(* IEC 61131-3 sources: Hal/Libraries/CAN_Lib, 3 files *)

(* ---- CAN_Lib.typ ---- *)
(********************************************************************
 * COPYRIGHT -- Bernecker + Rainer
 ********************************************************************
 * Library: CAN_Lib
 * File: CAN_Lib.typ
 * Author: B+R
 ********************************************************************
 * Data types of library CAN_Lib
 ********************************************************************)

TYPE
	INFO_typ : STRUCT				(*CAN statistic data*)
		received	: UDINT ;		(*the sum of all received CAN frames*)
		transmit	: UDINT ;		(*the sum of all sent CAN frames*)
		error	: UDINT ;			(*the sum of all error messages from the CAN device*)
		busoff	: UDINT ;			(*the sum of all CAN BusOff errors*)
		warning	: UDINT ;			(*the sum of all CAN warning errors*)
		other	: UDINT ;			(*the sum of other errors*)
		lost	: UDINT ;			(*the sum of all overwritten CAN frames*)
		stufferror	: UDINT ;		(*the sum of stuff errors*)
		formerror	: UDINT ;		(*the sum of form errors*)
		ackerror	: UDINT ;		(*the sum of ack errors*)
		bit1error	: UDINT ;		(*the sum of bit1 errors*)
		bit0error	: UDINT ;		(*the sum of bit0 errors*)
		crcerror	: UDINT ;		(*the sum of crc errors*)
		lec0	: UDINT ;			(*the sum of all errors with Last Error Code=0*)
		rxirq	: UDINT ;			(*the sum of all received interrupts*)
		txirq	: UDINT ;			(*the sum of all sent interrupts*)
	END_STRUCT;
	DevParam : STRUCT				(*points to the DeviceParameter structure*)
		baudrate	: USINT ;		(*baud rate for the CAN controller to be opened*)
		cob_nr	: UINT ;			(*number of communication objects*)
		pError	: UDINT ;			(*address of / pointer to the error variable*)
		pDevice	: UDINT ;			(*address of / pointer to the DeviceString*)
		info	: UINT ;			(*bit 7 = 1 enables extended mode for the controller*)
	END_STRUCT;
END_TYPE

(* ---- CAN_Lib.fun ---- *)
(********************************************************************
 * COPYRIGHT -- Bernecker + Rainer
 ********************************************************************
 * Library: CAN_Lib
 * File: CAN_Lib.fun
 * Author: B+R
 ********************************************************************
 * Functions and function blocks of library CAN_Lib
 ********************************************************************)

FUNCTION_BLOCK CANinfo			(*reads the statistical data from a CAN device*)
	VAR_INPUT
		enable	:BOOL;			(*enables execution*)
		us_ident	:UDINT;		(*us_ident identifier from CANopen*)
		info_adr	:UDINT;		(*pointer to the CANinfo structure INFO_typ*)
	END_VAR
	VAR_OUTPUT
		status	:UINT;			(*execution status: ERR_OK, ERR_FUB_ENABLE_FALSE, 0xXXXX = see help*)
	END_VAR
END_FUNCTION_BLOCK

FUNCTION_BLOCK CANMulQueue		(*installs a queue for multiple CAN identifiers in the read direction*)
	VAR_INPUT
		enable	:BOOL;			(*enables execution*)
		us_ident	:UDINT;		(*us_ident from CANopen / CANMulOpen*)
		pCAN_id	:UDINT;			(*pointer to an array of CAN identifiers*)
		ID_nr	:USINT;			(*number of CAN identifiers*)
		size	:UINT;			(*number of telegrams in the queue*)
	END_VAR
	VAR_OUTPUT
		q_ident	:UDINT;			(*identifier for CANmulrd*)
		status	:UINT;			(*execution status: ERR_OK, ERR_FUB_ENABLE_FALSE, 0xXXXX = see help*)
	END_VAR
	VAR
		old_enable	:BOOL;		(*internal variable*)
		cob_handle	:UDINT;		(*internal variable*)
		init_cnt	:UDINT;		(*internal variable*)
	END_VAR
END_FUNCTION_BLOCK

FUNCTION_BLOCK CANxMulQueue		(*installs a queue for multiple CAN identifiers in the read direction*)
	VAR_INPUT
		enable	:BOOL;			(*enables execution*)
		us_ident	:UDINT;		(*us_ident from CANopen / CANMulOpen*)
		pCAN_id	:UDINT;			(*pointer to an array of CAN identifiers*)
		ID_nr	:UDINT;			(*number of CAN identifiers*)
		size	:UINT;			(*number of telegrams in the queue*)
	END_VAR
	VAR_OUTPUT
		q_ident	:UDINT;			(*identifier for CANmulrd*)
		status	:UINT;			(*execution status: ERR_OK, ERR_FUB_ENABLE_FALSE, 0xXXXX = see help*)
	END_VAR
	VAR
		old_enable	:BOOL;		(*internal variable*)
		cob_handle	:UDINT;		(*internal variable*)
		init_cnt	:UDINT;		(*internal variable*)
	END_VAR
END_FUNCTION_BLOCK

FUNCTION_BLOCK CANMulOpen		(*initializes numerous CAN controllers and allocates the appropriate resources*)
	VAR_INPUT
		enable	:BOOL;			(*enables execution*)
		pDevParam	:UDINT;		(*pointer to the DeviceParameter structure*)
		dev_nr	:USINT;			(*number of CAN controllers to be opened*)
	END_VAR
	VAR_OUTPUT
		us_ident	:UDINT;		(*identifier for all additional CAN function blocks*)
		status	:UINT;			(*execution status: ERR_OK, ERR_FUB_ENABLE_FALSE, 0xXXXX = see help*)
	END_VAR
	VAR
		old_enable	:BOOL;		(*internal variable*)
		init_cnt	:UDINT;		(*internal variable*)
	END_VAR
END_FUNCTION_BLOCK

FUNCTION_BLOCK CANMulrd			(*copies data from the queue to the buffer or sends an error in the status*)
	VAR_INPUT
		enable	:BOOL;			(*enables execution*)
		q_ident	:UDINT;			(*identifier q_ident from CANMulQueue*)
		data_adr	:UDINT;		(*CAN data*)
	END_VAR
	VAR_OUTPUT
		size	:UINT;			(*length of the data*)
		ID	:UDINT;				(*CAN identifier which received the data*)
		status	:UINT;			(*execution status: ERR_OK, ERR_FUB_ENABLE_FALSE, 0xXXXX = see help*)
	END_VAR
END_FUNCTION_BLOCK

FUNCTION_BLOCK CANTime			(*reads the time stamp for a CAN object*)
	VAR_INPUT
		enable		:BOOL;		(*enables execution*)
		us_ident	:UDINT;		(*user ident from CANopen() / CANMulOpen()*)
		can_id	:UDINT;			(*CAN identifier*)
		pSystemTick	:UDINT;		(*pointer to the SystemTick counter*)
		pSystemStamp	:UDINT;	(*pointer to the SystemStamp*)
	END_VAR
	VAR_OUTPUT
		status	:UINT;			(*execution status: ERR_OK, ERR_FUB_ENABLE_FALSE, 0xXXXX = see help*)
	END_VAR
	VAR
		old_enable	:BOOL;		(*internal variable*)
		old_id	:UDINT;			(*internal variable*)
		cob_handle	:UDINT;		(*internal variable*)
	END_VAR
END_FUNCTION_BLOCK

FUNCTION_BLOCK CANquwr			(*sends a CAN message with the given CAN identifier to the CAN controller for transmission*)
	VAR_INPUT
		enable	:BOOL;			(*enables execution*)
		us_ident	:UDINT;		(*user ident number from the CANopen() function*)
		can_id	:UDINT;			(*CAN identifier*)
		data_adr	:UDINT;		(*address of the CAN data (max. 8 bytes)*)
		data_lng	:USINT;		(*length of the data (max. 8 bytes)*)
	END_VAR
	VAR_OUTPUT
		status	:UINT;			(*execution status: ERR_OK, ERR_FUB_ENABLE_FALSE, 0xXXXX = see help*)
	END_VAR
	VAR
		old_enable	:BOOL;		(*internal variable*)
		cob_handle	:UDINT;		(*internal variable*)
		init_cnt	:UDINT;		(*internal variable*)
	END_VAR
END_FUNCTION_BLOCK

FUNCTION_BLOCK SetNdNr			(*saves the transferred node number and device description in the CRM*)
	VAR_INPUT
		enable	:BOOL;			(*enables execution*)
		device	:UDINT;			(*pointer to a string containing the device description, e.g. "SLx.SSx.IFx"*)
		nodenr	:USINT;			(*new node number*)
	END_VAR
	VAR_OUTPUT
		status	:UINT;			(*execution status: ERR_OK, ERR_FUB_ENABLE_FALSE, 0xXXXX = see help*)
	END_VAR
END_FUNCTION_BLOCK

FUNCTION_BLOCK GetNdNr			(*reads the stored node number and device description from the CRM*)
	VAR_INPUT
		enable	:BOOL;			(*enables execution*)
		dev_adr	:UDINT;			(*pointer to a string containing the device description, e.g. "SLx.SSx.IFx"*)
	END_VAR
	VAR_OUTPUT
		nodenr	:USINT;			(*the node number read from the CRM*)
		status	:UINT;			(*execution status: ERR_OK, ERR_FUB_ENABLE_FALSE, 0xXXXX = see help*)
	END_VAR
END_FUNCTION_BLOCK

FUNCTION_BLOCK CMSexit			(*free the ressources of the list of CMS objects defined with the CMSinit() function*)
	VAR_INPUT
		enable	:BOOL;			(*enables execution*)
		cms_ident	:UDINT;		(*CMS identifier from CMSinit()*)
	END_VAR
	VAR_OUTPUT
		status	:UINT;			(*execution status: ERR_OK, ERR_FUB_ENABLE_FALSE, 0xXXXX = see help*)
	END_VAR
END_FUNCTION_BLOCK

FUNCTION_BLOCK CMSmain			(*edits the list of CMS objects defined with the CMSinit() function*)
	VAR_INPUT
		enable	:BOOL;			(*enables execution*)
		cms_ident	:UDINT;		(*CMS identifier from CMSinit()*)
		cms_mode	:UDINT;		(*2 ... WRITE, send/update data*)
	END_VAR
	VAR_OUTPUT
		status	:UINT;			(*execution status: ERR_OK, ERR_FUB_ENABLE_FALSE, 0xXXXX = see help*)
	END_VAR
	VAR
		init_cnt	:UDINT;		(*internal variable*)
	END_VAR
END_FUNCTION_BLOCK

FUNCTION_BLOCK CMSinit			(*sends and receives CMS objects*)
	VAR_INPUT
		enable	:BOOL;			(*enables execution*)
		us_ident	:UDINT;		(*user ident from CANopen()*)
		user_type	:USINT;		(*0 CLIENT node type, 1 SERVER node type*)
		queue_cnt	:UINT;		(*reserved*)
		modul_name	:UDINT;		(*pointer to the string containing the name of the data object*)
	END_VAR
	VAR_OUTPUT
		cms_entry	:UINT;		(*error entry number or number of CMS objects in the CMS data object*)
		cms_ident	:UDINT;		(*CMS identifier is needed for CMSmain()*)
		status	:UINT;			(*execution status: ERR_OK, ERR_FUB_ENABLE_FALSE, 0xXXXX = see help*)
	END_VAR
	VAR
		old_enable	:BOOL;		(*internal variable*)
		init_cnt	:UDINT;		(*internal variable*)
	END_VAR
END_FUNCTION_BLOCK

FUNCTION_BLOCK CMSdlreq			(*transfers a "multiplexed domain" object of any data size from the client to the server*)
	VAR_INPUT
		enable	:BOOL;			(*enables execution*)
		initiate	:BOOL;		(*pos. edge (0->1) ... Initiate new domain*)
		us_ident	:UDINT;		(*user ID from CANopen()*)
		client_id	:UDINT;		(*CAN identifier for the send COB from client to server*)
		server_id	:UDINT;		(*CAN identifier for the send COB from server to client*)
		mult	:UDINT;			(*multiplexer for multiplexed domain*)
		data_adr	:UDINT;		(*address of the download data*)
		data_len	:UDINT;		(*length of the download data*)
	END_VAR
	VAR_OUTPUT
		add_code	:UINT;		(*additional error information in the event of abnormal termination*)
		err_class	:USINT;		(*error class according to CANopen()*)
		err_code	:USINT;		(*error according to CANopen()*)
		dl_len	:UDINT;			(*size of the download data sent*)
		status	:UINT;			(*execution status: ERR_OK, ERR_FUB_ENABLE_FALSE, 0xXXXX = see help*)
	END_VAR
	VAR
		cob_handle	:UDINT;		(*internal variable*)
		init_cnt	:UDINT;		(*internal variable*)
		old_enable	:BOOL;		(*internal variable*)
	END_VAR
END_FUNCTION_BLOCK

FUNCTION_BLOCK CMSdlcon			(*enables a "multiplexed domain" object of any data length to be received by the server*)
	VAR_INPUT
		enable	:BOOL;			(*enables execution*)
		initiate	:BOOL;		(*1 ... startpulse, activation receiving the domain*)
		us_ident	:UDINT;		(*user ID from CANopen()*)
		client_id	:UDINT;		(*CAN identifier for the send COB from client to server*)
		server_id	:UDINT;		(*CAN identifier for the send COB from server to client*)
		data_adr	:UDINT;		(*address of the download data*)
		data_len	:UDINT;		(*length of the download data in bytes*)
	END_VAR
	VAR_OUTPUT
		add_code	:UINT;		(*additional error information in the event of abnormal termination*)
		err_class	:USINT;		(*error class according to CANopen()*)
		err_code	:USINT;		(*error according to CANopen()*)
		mult	:UDINT;			(*multiplexer for multiplexed domain*)
		dl_len	:UDINT;			(*size of the data already downloaded*)
		status	:UINT;			(*execution status: ERR_OK, ERR_FUB_ENABLE_FALSE, 0xXXXX = see help*)
	END_VAR
	VAR
		old_enable	:BOOL;		(*internal variable*)
		cob_handle	:UDINT;		(*internal variable*)
		init_cnt	:UDINT;		(*internal variable*)
	END_VAR
END_FUNCTION_BLOCK

FUNCTION_BLOCK CANxnode			(*determines the node number set with the x-th CAN node switch*)
	VAR_INPUT
		enable	:BOOL;			(*enables execution*)
		us_ident	:UDINT;		(*user Ident from CANopen()*)
	END_VAR
	VAR_OUTPUT
		node_nr	:USINT;			(*node number of the CAN station (0x00 through 0xFF)*)
		status	:UINT;			(*execution status: ERR_OK, ERR_FUB_ENABLE_FALSE, 0xXXXX = see help*)
	END_VAR
END_FUNCTION_BLOCK

FUNCTION_BLOCK CANwrite			(*sends a CAN message with the given CAN identifier to the CAN controller for transmission*)
	VAR_INPUT
		enable	:BOOL;			(*enables execution*)
		us_ident	:UDINT;		(*user ident number from the CANopen() function*)
		can_id	:UDINT;			(*CAN identifier*)
		data_adr	:UDINT;		(*address of the CAN data (max. 8 bytes)*)
		data_lng	:USINT;		(*length of the data (max. 8 bytes)*)
	END_VAR
	VAR_OUTPUT
		status	:UINT;			(*execution status: ERR_OK, ERR_FUB_ENABLE_FALSE, 0xXXXX = see help*)
	END_VAR
	VAR
		old_enable	:BOOL;		(*internal variable*)
		old_id	:UDINT;			(*internal variable*)
		cob_handle	:UDINT;		(*internal variable*)
		init_cnt	:UDINT;		(*internal variable*)
		wr_order	:USINT;		(*internal variable*)
		align_byte	:USINT;		(*internal variable*)
	END_VAR
END_FUNCTION_BLOCK

FUNCTION_BLOCK CANupd			(*gives the response to an RTR request telegram to the send node*)
	VAR_INPUT
		enable	:BOOL;			(*enables execution*)
		us_ident	:UDINT;		(*user ident from CANopen()*)
		can_id	:UDINT;			(*CAN identifier*)
		data_adr	:UDINT;		(*address of the data area in which the update data is stored*)
		data_lng	:USINT;		(*length of the update data in bytes*)
	END_VAR
	VAR_OUTPUT
		status	:UINT;			(*execution status: ERR_OK, ERR_FUB_ENABLE_FALSE, 0xXXXX = see help*)
	END_VAR
	VAR
		old_enable	:BOOL;		(*internal variable*)
		old_id	:UDINT;			(*internal variable*)
		cob_handle	:UDINT;		(*internal variable*)
		init_cnt	:UDINT;		(*internal variable*)
	END_VAR
END_FUNCTION_BLOCK

FUNCTION_BLOCK CANngp			(*handles the Node Guarding Protocol according to CAL on the NMT slave*)
	VAR_INPUT
		enable	:BOOL;			(*enables execution*)
		us_ident	:UDINT;		(*user ident from CANopen()*)
		can_id	:UDINT;			(*CAN identifier*)
		nd_state	:USINT;		(*node status*)
	END_VAR
	VAR_OUTPUT
		status	:UINT;			(*execution status: ERR_OK, ERR_FUB_ENABLE_FALSE, 0xXXXX = see help*)
	END_VAR
	VAR
		old_enable	:BOOL;		(*internal variable*)
		old_id	:UDINT;			(*internal variable*)
		cob_handle	:UDINT;		(*internal variable*)
		init_cnt	:UDINT;		(*internal variable*)
	END_VAR
END_FUNCTION_BLOCK

FUNCTION_BLOCK CANrwtab			(*edits the list of variables (variables table) defined with the CANdftab()*)
	VAR_INPUT
		enable	:BOOL;			(*enables execution*)
		tab_ident	:UDINT;		(*table identifier from CANdftab()*)
	END_VAR
	VAR_OUTPUT
		status	:UINT;			(*execution status: ERR_OK, ERR_FUB_ENABLE_FALSE, 0xXXXX = see help*)
	END_VAR
END_FUNCTION_BLOCK

FUNCTION_BLOCK CANrtr			(*sends an RTR request frame on the CAN bus*)
	VAR_INPUT
		enable	:BOOL;			(*enables execution*)
		request	:BOOL;			(*0 poll data buffer, 1 send RTR request*)
		us_ident	:UDINT;		(*user ident from CANopen()*)
		can_id	:UDINT;			(*CAN identifier*)
		data_adr	:UDINT;		(*address of the data area in which the data received is stored*)
	END_VAR
	VAR_OUTPUT
		data_lng	:USINT;		(*length of the received data in bytes*)
		status	:UINT;			(*execution status: ERR_OK, ERR_FUB_ENABLE_FALSE, 0xXXXX = see help*)
	END_VAR
	VAR
		old_enable	:BOOL;		(*internal variable*)
		cob_handle	:UDINT;		(*internal variable*)
		init_cnt	:UDINT;		(*internal variable*)
	END_VAR
END_FUNCTION_BLOCK

FUNCTION_BLOCK CANread			(*reads CAN messages from the CAN controller*)
	VAR_INPUT
		enable	:BOOL;			(*enables execution*)
		us_ident	:UDINT;		(*user ident number from the CANopen() function*)
		can_id	:UDINT;			(*CAN identifier*)
		data_adr	:UDINT;		(*address where the read data is stored (max. 8 bytes)*)
	END_VAR
	VAR_OUTPUT
		data_lng	:USINT;		(*length of the data*)
		status	:UINT;			(*execution status: ERR_OK, ERR_FUB_ENABLE_FALSE, 0xXXXX = see help*)
	END_VAR
	VAR
		old_enable	:BOOL;		(*internal variable*)
		cob_handle	:UDINT;		(*internal variable*)
		init_cnt	:UDINT;		(*internal variable*)
	END_VAR
END_FUNCTION_BLOCK

FUNCTION_BLOCK CANrd			(*copies data from the queue to the buffer or sends an error in the status*)
	VAR_INPUT
		enable	:BOOL;			(*enables execution*)
		q_ident	:UDINT;			(*queue identifier from CANqueue()*)
		data_adr	:UDINT;		(*address of the data area where CAN data from the receive queue is stored*)
	END_VAR
	VAR_OUTPUT
		size	:UINT;			(*length of the CAN data in bytes*)
		status	:UINT;			(*execution status: ERR_OK, ERR_FUB_ENABLE_FALSE, 0xXXXX = see help*)
	END_VAR
END_FUNCTION_BLOCK

FUNCTION_BLOCK CANxrd			(*copies data from the queue to the buffer or sends an error in the status*)
	VAR_INPUT
		enable	:BOOL;			(*enables execution*)
		q_ident	:UDINT;			(*queue identifier from CANqueue()*)
		data_adr	:UDINT;		(*address of the data area where CAN data from the receive queue is stored*)
	END_VAR
	VAR_OUTPUT
		can_id	:UDINT;			(*CAN identifier*)
		size	:UINT;			(*length of the CAN data in bytes*)
		status	:UINT;			(*execution status: ERR_OK, ERR_FUB_ENABLE_FALSE, 0xXXXX = see help*)
	END_VAR
END_FUNCTION_BLOCK

FUNCTION_BLOCK CANqueue			(*installs a queue for a CAN identifier in the read direction*)
	VAR_INPUT
		enable	:BOOL;			(*enables execution*)
		us_ident	:UDINT;		(*user Ident from CANopen()*)
		can_id	:UDINT;			(*CAN identifier for the queue*)
		size	:UINT;			(*number of telegrams in the queue*)
	END_VAR
	VAR_OUTPUT
		q_ident	:UDINT;			(*queue identifier for the CANrd()*)
		status	:UINT;			(*execution status: ERR_OK, ERR_FUB_ENABLE_FALSE, 0xXXXX = see help*)
	END_VAR
	VAR
		old_enable	:BOOL;		(*internal variable*)
		cob_handle	:UDINT;		(*internal variable*)
		init_cnt	:UDINT;		(*internal variable*)
	END_VAR
END_FUNCTION_BLOCK

FUNCTION_BLOCK CANopen			(*initializes the CAN controller and requests the necessary resources (e.g. memory)*)
	VAR_INPUT
		enable	:BOOL;			(*enables execution*)
		baud_rate	:USINT;		(*baud rate at which the CAN interface should be operated*)
		cob_anz	:UINT;			(*max. permissible number of COBs (communication objects)*)
		error_adr	:UDINT;		(*pointer to an error variable, e.g. Bit 15 = 1 the CAN bus is in the BusOff state*)
		device	:UDINT;			(*address of a string which clearly describes the CAN interface*)
		info	:UINT;			(*enables/disables extended mode for the CAN controller*)
	END_VAR
	VAR_OUTPUT
		us_ident	:UDINT;		(*is required for the other functions of the CAN_Lib library in order to identify a CAN interface clearly*)
		status	:UINT;			(*execution status: ERR_OK, ERR_FUB_ENABLE_FALSE, 0xXXXX = see help*)
	END_VAR
	VAR
		old_enable	:BOOL;		(*internal variable*)
		init_cnt	:UDINT;		(*internal variable*)
	END_VAR
END_FUNCTION_BLOCK

FUNCTION_BLOCK CANnode			(*determines the CAN node number*)
	VAR_INPUT
		enable	:BOOL;			(*enables execution*)
	END_VAR
	VAR_OUTPUT
		node_nr	:USINT;			(*node number of the CAN station (0x00 through 0xFF)*)
		status	:UINT;			(*execution status: ERR_OK, ERR_FUB_ENABLE_FALSE, 0xXXXX = see help*)
	END_VAR
END_FUNCTION_BLOCK

FUNCTION_BLOCK CANgetid			(*confirms the CAN identifier which the exception trigged in the context of an exception object*)
	VAR_INPUT
		enable	:BOOL;			(*enables execution*)
		data_adr	:UDINT;		(*address of the data area in which the data received is stored*)
	END_VAR
	VAR_OUTPUT
		data_lng	:USINT;		(*length of the received data in bytes*)
		can_id	:UDINT;			(*CAN identifier for the exception*)
		status	:UINT;			(*execution status: ERR_OK, ERR_FUB_ENABLE_FALSE, 0xXXXX = see help*)
	END_VAR
	VAR
		init_cnt	:UDINT;		(*internal variable*)
	END_VAR
END_FUNCTION_BLOCK

FUNCTION_BLOCK CANexcep			(*activates a pre-installed exception object with the exception number exc_no*)
	VAR_INPUT
		enable	:BOOL;			(*enables execution*)
		us_ident	:UDINT;		(*user Ident from CANopen()*)
		can_id	:UDINT;			(*CAN identifier*)
		exc_nr	:USINT;			(*number of the exception (exception numbers 208 to 223 are reserved for CAN)*)
	END_VAR
	VAR_OUTPUT
		status	:UINT;			(*execution status: ERR_OK, ERR_FUB_ENABLE_FALSE, 0xXXXX = see help*)
	END_VAR
	VAR
		old_enable	:BOOL;		(*internal variable*)
		init_cnt	:UDINT;		(*internal variable*)
		cob_handle	:UDINT;		(*internal variable*)
		ex_p	:UDINT;			(*internal variable*)
		ex_maxtask	:UDINT;		(*internal variable*)
		ss_irqvw_p	:UDINT;		(*internal variable*)
	END_VAR
END_FUNCTION_BLOCK

FUNCTION_BLOCK CANdftab			(*supplies a variables list (variables table) defined by the user with data about the CAN bus*)
	VAR_INPUT
		enable	:BOOL;			(*enables execution*)
		us_ident	:UDINT;		(*user ident number from the CANopen() function*)
		table_adr	:UDINT;		(*address of the variables table*)
		tab_num	:UINT;			(*number of entries in the variables table*)
	END_VAR
	VAR_OUTPUT
		tab_ident	:UDINT;		(*table identifier for CANrwtab()*)
		status	:UINT;			(*execution status: ERR_OK, ERR_FUB_ENABLE_FALSE, 0xXXXX = see help*)
	END_VAR
	VAR
		old_enable	:BOOL;		(*internal variable*)
		init_cnt	:UDINT;		(*internal variable*)
	END_VAR
END_FUNCTION_BLOCK

FUNCTION_BLOCK CANbtreg			(*configures a special bit timing register values for the CAN controller (Intel 82527)*)
	VAR_INPUT
		enable	:BOOL;			(*enables execution*)
		us_ident	:UDINT;		(*user Ident from CANopen()*)
		treg0	:UDINT;			(*bit timing register 0*)
		treg1	:UDINT;			(*bit timing Register 1*)
	END_VAR
	VAR_OUTPUT
		status	:UINT;			(*execution status: ERR_OK, ERR_FUB_ENABLE_FALSE, 0xXXXX = see help*)
	END_VAR
END_FUNCTION_BLOCK

(* ---- CAN_Lib.var ---- *)
(********************************************************************
 * COPYRIGHT (C) BERNECKER + RAINER, AUSTRIA, A-5142 EGGELSBERG
 ********************************************************************
 * Library: CAN_Lib
 * File: CAN_Lib.var
 * Created: 22.02.2010
 ********************************************************************
 * Constants of library CAN_Lib
 ********************************************************************)
VAR CONSTANT
	canERR_CAN_NOENTRY		: UINT	:= 8800;		(*not enough communication objects (COBs) available as specified in CANopen*)
	canERR_CAN_NOMEM		: UINT	:= 8801;		(*not enough memory available for resources*)
	canERR_CAN_WRIDENT		: UINT	:= 8802;		(*wrong identifier*)
	canERR_CAN_COBUSED		: UINT	:= 8803;		(*communication objects (COBs) identifier is already being used in the system*)
	canERR_CAN_WRCANID		: UINT	:= 8804;		(*wrong CAN identifier: Only standard CAN identifiers (11 bits) up to 2047 are permitted*)
	canERR_CAN_WRUSERID		: UINT	:= 8805;		(*incorrect user ID us_ident transferred, or the FBK cannot be used after a CANMulOpen*)
	canERR_CAN_COBDEF		: UINT	:= 8806;		(*a COB with the specified CAN identifier has already been defined in the system*)
	canERR_CAN_WRDEF		: UINT	:= 8807;		(*false CAN identifier definition*)
	canERR_CAN_WRHDLE		: UINT	:= 8808;		(*COB management (FBK memory) destroyed*)
	canERR_CAN_BUSY			: UINT	:= 8809;		(*CAN operation with the same CAN identifier is busy*)
	canERR_CAN_QFULL		: UINT	:= 8810;		(*transmit queue full*)
	canERR_CAN_BUSOFF		: UINT	:= 8811;		(*CAN bus is BusOff. Different baud rate on different nodes?*)
	canERR_CAN_NOHIGH		: UINT	:= 8812;		(*no more buffers available: All buffers (max. 13) in the can controller have already been defined and assigned*)
	canERR_CAN_NOTINST		: UINT	:= 8813;		(*CAN driver not installed: CAN2000.BR not loaded (needs to be transferred to target system)*)
	canERR_CAN_WRLNG		: UINT	:= 8814;		(*data type of event PV is not BYTES or the length of a write PV is greater than 8 bytes: CAN FBKs can only send data of length 8 bytes to the CAN bus*)
	canERR_CAN_BDRATE		: UINT	:= 8815;		(*illegal baud rate *)
	canERR_CAN_COBANZ		: UINT	:= 8816;		(*cob_anz in CANopen/CANMulOpen incorrect: cob_no must be less than 2048 and greater than 0*)
	canERR_CAN_NOCONTR		: UINT	:= 8817;		(*no CAN controller found: Error in the device string of the FBK CANopen / CANMulOpen or the CAN controller is not ready - hardware may not be present*)
	canERR_CAN_HTLXINF		: UINT	:= 8818;		(*error analyzing hardware*)
	canERR_CAN_HTLQUIT		: UINT	:= 8819;		(*error in interrupt handling*)
	canERR_CAN_NOFUNC		: UINT	:= 8820;		(*error in interrupt handling*)
	canERR_CAN_WRUSRTYP		: UINT	:= 8821;		(*user_typ in CMSinit is incorrect: user_typ must be 0 for client or 1 for server*)
	canERR_WRCMSOBJ			: UINT	:= 8822;		(*CMS object incorrectly defined: Syntax error in the CMS data object for CMSinit() (see cms_entry)*)
	canERR_CAN_WRSTRUCT		: UINT	:= 8823;		(*invalid CMS structure: The structure is too complex (only simple structures are permitted)*)
	canERR_CAN_WRMODE		: UINT	:= 8824;		(*incorrect value for cms_mode transferred to the CMSmain() function (valid value: 2)*)
	canERR_CAN_NO_NODE		: UINT	:= 8825;		(*node number cannot be read*)
	canERR_CAN_NILPTR		: UINT	:= 8826;		(*an invalid parameter has been transferred (NULL)*)
	canERR_CAN_IRQHANDLE	: UINT	:= 8827;		(*internal management is destroyed in the interrupt handler*)
	canERR_CAN_ABORTED		: UINT	:= 8828;		(*abort protocol has been sent to the client (>add_code)*)
	canERR_CAN_ABORTRECEIV	: UINT	:= 8829;		(*abort protocol has been received from the client*)
	canERR_CAN_FBHANDLE		: UINT	:= 8830;		(*incorrect FBCAN handle*)
	canERR_CAN_EXTENDED		: UINT	:= 8831;		(*conflict with standard/extended mode (11 or 29-bit CAN identifier): FBK configuration and system configuration (Automation Studio) of CAN interface do not match*)
	canERR_CMS_MULTIPLEX	: UINT	:= 8832;		(*CMS multiplexer definition error: Different object_typ, access_typ or ID or a multiplexer has been used more than once for an ID*)
	canERR_CAN_WROBJ		: UINT	:= 8833;		(*CAN object error: Tried to use a dynamic PV. Use a normal PV*)
	canERR_CAN_BITMODE		: UINT	:= 8834;		(*CAN identifier mode configured differently (11-bit / 29-bit, see the Automation Studio CAN device configuration)*)
	canERR_FBCAN_COB		: UINT	:= 8837;		(*INA2000 CAN: COB not defined*)
	canERR_FBCAN_NODENR		: UINT	:= 8838;		(*INA2000 CAN: Node number too large*)
	canERR_FBCAN_HANDLE		: UINT	:= 8839;		(*INA2000 CAN: Incorrect handle*)
	canERR_FBCAN_RXBUF		: UINT	:= 8840;		(*INA2000 CAN: No Rx buffer free*)
	canERR_CAN_STUFF		: UINT	:= 8841;		(*Warning: CAN: Stuff error -> CAN ID collision / baud rate*)
	canERR_CAN_FORM			: UINT	:= 8842;		(*Warning: CAN: Format error -> Baud rate*)
	canERR_CAN_ACK			: UINT	:= 8843;		(*Warning: CAN: ACK error - No acknowledge from other nodes*)
	canERR_CAN_BIT1			: UINT	:= 8844;		(*Warning: CAN: Bit1 send error (recessive bit)*)
	canERR_CAN_BIT0			: UINT	:= 8845;		(*Warning: CAN: Bit0 send error (dominant bit)*)
	canERR_CAN_CRC			: UINT	:= 8846;		(*Warning: CAN: CRC checksum error*)
	canERR_WRONG_OBJNR		: UINT	:= 8850;		(*CAN CCI: Object number not within value range*)
	canERR_NO_INIT_STATE	: UINT	:= 8851;		(*CAN CCI: Error during initialization*)
	canERR_NO_BUSOFF_STATE	: UINT	:= 8852;		(*CAN CCI: BUS_OFF problem*)
	canERR_NO_BUFFER_CFG	: UINT	:= 8853;		(*CAN CCI: Buffer not configured*)
	canERR_HW_RESET_ACTIVE	: UINT	:= 8854;		(*CAN CCI: Hardware in reset state*)
	canERR_CPU_UPDATE		: UINT	:= 8855;		(*CAN CCI: Error updating data*)
	canERR_OBJ_ACTIVE		: UINT	:= 8856;		(*CAN CCI: Buffer being processed*)
	canERR_READ_ONLY_OBJ	: UINT	:= 8857;		(*CAN CCI: Read-only object*)
	canERR_WRONG_CAN_MODE	: UINT	:= 8858;		(*CAN CCI: Incorrect mode (Standard/Extended)*)
	canERR_WRONG_MSG_LEN	: UINT	:= 8859;		(*the specified length does not match the length of the CAN message*)
	canERR_TXIE_NOT_ALLOWED	: UINT	:= 8860;		(*CAN CCI: Transmit interrupt not allowed*)
	canERR_TXIE_ALLOWED		: UINT	:= 8861;		(*CAN CCI: Transmit interrupt has to be set*)
	canERR_RXIE_NOT_ALLOWED	: UINT	:= 8862;		(*CAN CCI: Receive interrupt not allowed*)
	canERR_RXIE_ALLOWED		: UINT	:= 8863;		(*CAN CCI: Receive interrupt has to be set*)
	canERR_WRONG_CAN_ID		: UINT	:= 8864;		(*CAN CCI: Incorrect CAN ID entered*)
	canERR_NO_RD_MODE		: UINT	:= 8865;		(*CAN CCI: Reading with send object*)
	canERR_NO_WR_MODE		: UINT	:= 8866;		(*CAN CCI: Writing with receive object*)
	canERR_NO_STATE_BOFF	: UINT	:= 8867;		(*CAN CCI: BUS_OFF state not accepted*)
	canERR_NO_STATE_INIT	: UINT	:= 8868;		(*CAN CCI: Init state not accepted*)
	canERR_NO_STATE_BON		: UINT	:= 8869;		(*CAN CCI: BUS_ON state not accepted*)
	canERR_NORMAL_NOT_POSIBLE:UINT	:= 8870;		(*CAN CCI: Interrupt number not allowed*)
	canERR_STATUS			: UINT	:= 8871;		(*CAN CCI: Error in status (structure)*)
	canERR_MSG_LOST			: UINT	:= 8872;		(*message lost: One or more data frames have been lost for this CAN identifier. The buffer has been overwritten but the data is consistent*)
	canERR_MAXRETRY_DATENINKONSIST : UINT	:= 8873;		(*CAN CCI: Read data inconsistent despite max. retries*)
	canERR_MAX_RETRY_CNT	: UINT	:= 8874;		(*CAN CCI: Retry counter expired*)
	canERR_DATEN_INKONSISTENT:UINT	:= 8875;		(*the data for this CAN identifier is inconsistent (new data received during CANread())*)
	canERR_NO_OBJ_FREE		: UINT	:= 8876;		(*send buffer is not free: This error occurs if a high-priority object has been defined without overwrite mode, for example, and the data from the last CMSmain() instruction is still in the CAN controller waiting to be sent*)
	canERR_NO_DATA			: UINT	:= 8877;		(*no current data available for the specified CAN identifier*)
END_VAR
